// TIA Portal V20 export
FUNCTION_BLOCK "FB_ManualControl"   // FB37, LAD
// stored: Access Published, MemoryReserve 100, Namespace Global, SetENOAutomatically false
   VAR RETAIN
      "Counter" { S7_SetPoint := 'True'} : CTU_INT;
   END_VAR
BEGIN

REGION Network 1
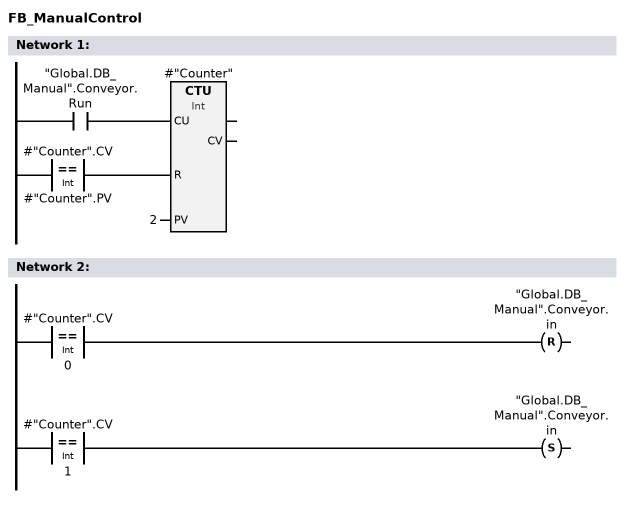
   RUNG wire#powerrail
      Contact( "Global.DB_Manual".Conveyor.Run )
      { S7_Templates := "value_type := Int" } #"Counter".CTU(r := wire#w1, pv := 2, cv =>)
   END_RUNG
   RUNG wire#powerrail
      { S7_Templates := "SrcType := Int" } EQ_Contact(in1 := #"Counter".CV, in2 := #"Counter".PV)
   END_RUNG wire#w1
   // the same network as SCL:
   #"Counter"(CU := "Global.DB_Manual".Conveyor.Run, R := #"Counter".CV = #"Counter".PV, PV := 2);   // CTU
END_REGION

REGION Network 2
   RUNG wire#powerrail
      { S7_Templates := "SrcType := Int" } EQ_Contact(in1 := #"Counter".CV, in2 := 0)
      R_Coil( "Global.DB_Manual".Conveyor.in )
   END_RUNG
   RUNG wire#powerrail
      { S7_Templates := "SrcType := Int" } EQ_Contact(in1 := #"Counter".CV, in2 := 1)
      S_Coil( "Global.DB_Manual".Conveyor.in )
   END_RUNG
   // the same network as SCL:
   IF #"Counter".CV = 0 THEN "Global.DB_Manual".Conveyor.in := FALSE; END_IF;
   IF #"Counter".CV = 1 THEN "Global.DB_Manual".Conveyor.in := TRUE; END_IF;
END_REGION
END_FUNCTION_BLOCK
